TYPE E_ModeLanguage :
(
	Deutsch := 1,
	English := 2
);
END_TYPE

(* stored: Version 1.1.0.1
   DUT E_ModeLanguage: Id {69005972-a676-4fe9-b262-de574ddbac92} *)
